PROGRAM OOPSDevelopmentTest
VAR
END_VAR

END_PROGRAM

(* stored: Version 1.1.0.1, ProductVersion 3.1.4024.12
   POU OOPSDevelopmentTest: Id {b8b13482-a341-41a8-a742-dcdb3e682f2a}, SpecialFunc None *)
